(* IEC 61131-3 sources: ics/BLR101_ProenixContact/BLR101_5_ILC171_44/LogicalPOUs/MISC, 2 files *)

(* ---- TICK_100MS.ST ---- *)
(*@PROPERTIES_EX@
TYPE: POU
LOCALE: 0
IEC_LANGUAGE: ST
PLC_TYPE: independent
PROC_TYPE: independent
GROUP: MISC
*)
(*@KEY@:DESCRIPTION*)

(*@KEY@:END_DESCRIPTION*)
PROGRAM TICK_100MS

(*Group:Default*)

VAR
	R_TRIG_1 :	R_TRIG;
END_VAR

VAR_EXTERNAL
	TICK_100MS :	BOOL;
	TICK_100MS_PLS :	BOOL;
END_VAR

(*@KEY@: WORKSHEET
NAME: TICK_100MS
IEC_LANGUAGE: ST
*)
TICK_100MS:= not TICK_100MS;

R_TRIG_1(CLK:=TICK_100MS);
TICK_100MS_PLS:=R_TRIG_1.Q;

(*@KEY@: END_WORKSHEET *)
END_PROGRAM

(* ---- TICK_1S.ST ---- *)
(*@PROPERTIES_EX@
TYPE: POU
LOCALE: 0
IEC_LANGUAGE: ST
PLC_TYPE: independent
PROC_TYPE: independent
GROUP: MISC
*)
(*@KEY@:DESCRIPTION*)

(*@KEY@:END_DESCRIPTION*)
PROGRAM TICK_1S

(*Group:Default*)

VAR_EXTERNAL
	TICK_1S :	BOOL;
END_VAR

VAR
	R_TRIG_1 :	R_TRIG;
END_VAR

VAR_EXTERNAL
	TICK_1S_PLS :	BOOL;
END_VAR

(*@KEY@: WORKSHEET
NAME: TICK_1S
IEC_LANGUAGE: ST
*)
TICK_1S:= not TICK_1S;

R_TRIG_1(CLK:= TICK_1S);
TICK_1S_PLS:=R_TRIG_1.Q;

(*@KEY@: END_WORKSHEET *)
END_PROGRAM
